// TIA Portal V17 export
// export: Created 2026-04-13T11:12:43.2392843Z, ExportSetting WithDefaults, DisplayName Totally Integrated Automation Portal, DisplayVersion V17 Update 4, DisplayName TIA Portal Openness, DisplayVersion V17 Update 4, DisplayName TIA Portal Version Control Interface, DisplayVersion V17, DisplayName SINAMICS Startdrive Advanced, DisplayVersion V17, DisplayName SINAMICS Startdrive G130, G150, S120, S150, SINAMICS MV, S210, DisplayVersion V17, DisplayName SINAMICS Startdrive G110M, G120, G120C, G120D, G120P, G115D, DisplayVersion V17, DisplayName STEP 7 Professional, DisplayVersion V17 Update 4, DisplayName STEP 7 Safety, DisplayVersion V17, DisplayName WinCC Professional, DisplayVersion V17 Update 4
FUNCTION_BLOCK "7-PID仿真LSim_PT3"   // FB80, SCL
{ S7_Optimized_Access := 'TRUE' }
VERSION : 2.1
// stored: AutoNumber true, IsIECCheckEnabled false, IsRetainMemResEnabled false, MemoryReserve 100, SetENOAutomatically false, UDAEnableTagReadback false
   VAR_INPUT
      input : Real;   // input variable
      tmLag1 : Real := 29.0;   // time lag 1 in s
      tmLag2 : Real := 17.5;   // time lag 2 in s
      tmLag3 : Real := 3.1;   // time lag 3 in s
      gain : Real := 1.0;   // proportional gain
      disturb : Real;   // disturbance variable (additional to "input")
      cycle : Real := 0.1;   // sample time [in sec]
      reset : Bool;   // complete restart (#output = #input)
   END_VAR
   VAR_OUTPUT
      error : Bool;   // error (#tmLag1 <= 0 or #tmLag2 <= 0 or #tmLag3 <= 0)
      status : Word;   // status (if #error = TRUE then status = 16#8001)
      output : Real;   // output signal (if #error = FALSE)
   END_VAR
   VAR
      statFback1 : Real;   // feedback path value 1
      statFback2 : Real;   // feedback path value 2
      statFback3 : Real;   // feedback path value 3
   END_VAR
   VAR_TEMP
      tempHvar : Real;   // help variable
      tempCycleR : Real;   // cycle to real
      tempTmLag1R : Real;   // time lag 1 to real
      tempTmLag2R : Real;   // time lag 2 to real
      tempTmLag3R : Real;   // time lag 3 to real
      tempOutvNew : Real;   // new output variable
   END_VAR
BEGIN
   //=============================================================================
   //SIEMENS AG
   //(c)Copyright 2017 All Rights Reserved
   //-----------------------------------------------------------------------------
   //Library:       Library for Controlled System Simulation
   //Tested with:   S7-1500 FW V2.0 / S7-1200 FW V4.2
   //Engineering:   STEP 7 V14 Upd2 (TIA Portal)
   //Restrictions:  Cyclic interrupt
   //Requirements:  memory card needed for S7-1500
   //Functionality: Simulation of an PT3-system
   //
   //                               gain
   //  F(p) = ------------------------------------------------------
   //         (tmLag1 * p + 1) * (tmLag2 * p + 1) * (tmLag3 * p + 1)
   //          
   //  Call the simulation in a cyclic interrupt with
   //  cyclic interrupt time at least = tmLag1/10!
   //-----------------------------------------------------------------------------
   //Change log table:
   //Version  Date       Expert in charge                Changes applied
   //02.00.00 03.02.2016 Siemens Industry Online Support Release (STEP 7 V13 SP1)
   //02.00.01 02.03.2017 Siemens Industry Online Support Release (STEP 7 V14)
   //=============================================================================
   // check parameter
   IF #tmLag1 <= 0 OR #tmLag2 <= 0 OR #tmLag3 <= 0 THEN
     #error := TRUE;
     #status := W#16#8001;     // Parameter Error
     #output := #input; //write output data
     #statFback1 := #input; //write static data
     #statFback2 := #input;
     #statFback3 := #input;
     RETURN;
   ELSE
     #error := FALSE;
     #status := W#16#0000;     // no error
   END_IF;

   IF #reset THEN //complete restart routine

     #output := #input;//write output data
     #statFback1 := #input;//write static data
     #statFback2 := #input;
     #statFback3 := #input;

   ELSE //cycle mode routine

     #tempCycleR  := #cycle*1000; //transform data type
     #tempTmLag1R := #tmLag1*1000;
     #tempTmLag2R := #tmLag2*1000;
     #tempTmLag3R := #tmLag3*1000;

     IF #tempCycleR * 0.5 > #tempTmLag1R THEN //limit TM_LAG1
       #tempTmLag1R := #tempCycleR * 0.5;
     END_IF;

     IF #tempCycleR * 0.5 > #tempTmLag2R THEN //limit TM_LAG2
       #tempTmLag2R := #tempCycleR * 0.5;
     END_IF;

     IF #tempCycleR * 0.5 > #tempTmLag3R THEN //limit TM_LAG2
       #tempTmLag3R := #tempCycleR * 0.5;
     END_IF;

     //1. first order lag algorithm
     #tempHvar     := #tempCycleR / (#tempTmLag1R * 2.0); 
     #tempHvar     := (#gain * (#input + #disturb) - #statFback1) * #tempHvar / (#tempHvar + 1.0);
     #tempOutvNew  := #tempHvar + #statFback1;
     #statFback1  := #tempHvar * 2.0 + #statFback1;

     //2. first order lag algorithm
     #tempHvar     := #tempCycleR / (#tempTmLag2R * 2.0); 
     #tempHvar     := ((#tempOutvNew - #statFback2) * #tempHvar) / (#tempHvar + 1.0);
     #tempOutvNew  := #tempHvar + #statFback2;
     #statFback2  := #tempHvar * 2.0 + #statFback2;

     //3. first order lag algorithm
     #tempHvar     := #tempCycleR / (#tempTmLag3R * 2.0); 
     #tempHvar     := ((#tempOutvNew - #statFback3) * #tempHvar) / (#tempHvar + 1.0);
     #tempOutvNew  := #tempHvar + #statFback3;
     #statFback3  := #tempHvar * 2.0 + #statFback3;

     #output := #tempOutvNew; //write output

   END_IF;
END_FUNCTION_BLOCK
